KUKA KRL data list: GlobalPosn.dat

&ACCESS RVO1
&REL 1
&PARAM EDITMASK = *
&PARAM TEMPLATE = C:\KRC\Roboter\Template\submit
DEFDAT GlobalPosn PUBLIC
; **************************************
; * Package:     TeslaCore             *
; * Release      V4.0.0                *
; * File:        GlobalPosn.dat        *
; * Date:        07.2016               *
; * GUI Version: > = V8.3              *
; **************************************

;FOLD Control Information
DECL GLOBAL INT nMaxGlobalPosn=10 ; Maximum # of global positions
GLOBAL STRUC PosnCtrl_Typ CHAR Comment[24], BOOL PosnEnabled,AtPosn, INT OutputCtrl, REAL A1_Tol, A2_Tol, A3_Tol, A4_Tol, A5_Tol, A6_Tol, E1_Tol, E2_Tol, E3_Tol, E4_Tol, E5_Tol, E6_Tol
DECL GLOBAL PosnCtrl_Typ xGP_Ctrl[10]
xGP_Ctrl[1]={Comment[]" ", PosnEnabled FALSE, AtPosn FALSE, OutputCtrl 0, A1_Tol 2.0, A2_Tol 2.0, A3_Tol 2.0, A4_Tol 2.0, A5_Tol 2.0, A6_Tol 2.0, E1_Tol 2.0, E2_Tol 2.0, E3_Tol 2.0, E4_Tol 2.0, E5_Tol 2.0, E6_Tol 2.0}
xGP_Ctrl[2]={Comment[]" ", PosnEnabled FALSE, AtPosn FALSE,OutputCtrl 0, A1_Tol 2.0, A2_Tol 2.0, A3_Tol 2.0, A4_Tol 2.0, A5_Tol 2.0, A6_Tol 2.0, E1_Tol 2.0, E2_Tol 2.0, E3_Tol 2.0, E4_Tol 2.0, E5_Tol 2.0, E6_Tol 2.0}
xGP_Ctrl[3]={Comment[]" ", PosnEnabled FALSE, AtPosn FALSE,OutputCtrl 0, A1_Tol 2.0, A2_Tol 2.0, A3_Tol 2.0, A4_Tol 2.0, A5_Tol 2.0, A6_Tol 2.0, E1_Tol 2.0, E2_Tol 2.0, E3_Tol 2.0, E4_Tol 2.0, E5_Tol 2.0, E6_Tol 2.0}
xGP_Ctrl[4]={Comment[]" ", PosnEnabled FALSE, AtPosn FALSE,OutputCtrl 0, A1_Tol 2.0, A2_Tol 2.0, A3_Tol 2.0, A4_Tol 2.0, A5_Tol 2.0, A6_Tol 2.0, E1_Tol 2.0, E2_Tol 2.0, E3_Tol 2.0, E4_Tol 2.0, E5_Tol 2.0, E6_Tol 2.0}
xGP_Ctrl[5]={Comment[]" ", PosnEnabled FALSE, AtPosn FALSE,OutputCtrl 0, A1_Tol 2.0, A2_Tol 2.0, A3_Tol 2.0, A4_Tol 2.0, A5_Tol 2.0, A6_Tol 2.0, E1_Tol 2.0, E2_Tol 2.0, E3_Tol 2.0, E4_Tol 2.0, E5_Tol 2.0, E6_Tol 2.0}
xGP_Ctrl[6]={Comment[]" ", PosnEnabled FALSE, AtPosn FALSE,OutputCtrl 0, A1_Tol 2.0, A2_Tol 2.0, A3_Tol 2.0, A4_Tol 2.0, A5_Tol 2.0, A6_Tol 2.0, E1_Tol 2.0, E2_Tol 2.0, E3_Tol 2.0, E4_Tol 2.0, E5_Tol 2.0, E6_Tol 2.0}
xGP_Ctrl[7]={Comment[]" ", PosnEnabled FALSE, AtPosn FALSE,OutputCtrl 0, A1_Tol 2.0, A2_Tol 2.0, A3_Tol 2.0, A4_Tol 2.0, A5_Tol 2.0, A6_Tol 2.0, E1_Tol 2.0, E2_Tol 2.0, E3_Tol 2.0, E4_Tol 2.0, E5_Tol 2.0, E6_Tol 2.0}
xGP_Ctrl[8]={Comment[]" ", PosnEnabled FALSE, AtPosn FALSE,OutputCtrl 0, A1_Tol 2.0, A2_Tol 2.0, A3_Tol 2.0, A4_Tol 2.0, A5_Tol 2.0, A6_Tol 2.0, E1_Tol 2.0, E2_Tol 2.0, E3_Tol 2.0, E4_Tol 2.0, E5_Tol 2.0, E6_Tol 2.0}
xGP_Ctrl[9]={Comment[]" ", PosnEnabled FALSE, AtPosn FALSE,OutputCtrl 0, A1_Tol 2.0, A2_Tol 2.0, A3_Tol 2.0, A4_Tol 2.0, A5_Tol 2.0, A6_Tol 2.0, E1_Tol 2.0, E2_Tol 2.0, E3_Tol 2.0, E4_Tol 2.0, E5_Tol 2.0, E6_Tol 2.0}
xGP_Ctrl[10]={Comment[]" ", PosnEnabled FALSE, AtPosn FALSE,OutputCtrl 0, A1_Tol 2.0, A2_Tol 2.0, A3_Tol 2.0, A4_Tol 2.0, A5_Tol 2.0, A6_Tol 2.0, E1_Tol 2.0, E2_Tol 2.0, E3_Tol 2.0, E4_Tol 2.0, E5_Tol 2.0, E6_Tol 2.0}
;ENDFOLD (Control Information)
;FOLD Positional Information
DECL GLOBAL E6AXIS XGlobal1={A1 0.0,A2 -90.0,A3 90.0,A4 0.0,A5 0.0,A6 0.0,E1 0.0,E2 0.0,E3 0.0,E4 0.0,E5 0.0,E6 0.0}
DECL GLOBAL FDAT FGlobal1={TOOL_NO 1,BASE_NO 0,IPO_FRAME #BASE,POINT2[] " ",TQ_STATE FALSE}
DECL GLOBAL PDAT PGlobal1={VEL 100.000,ACC 100.000,APO_DIST 100.000,GEAR_JERK 50.0000}
DECL GLOBAL LDAT LCGlobal1={VEL 2.00000,ACC 100.000,APO_DIST 100.000,APO_FAC 50.0000,AXIS_VEL 100.000,AXIS_ACC 100.000,ORI_TYP #VAR,CIRC_TYP #BASE,JERK_FAC 50.0000,GEAR_JERK 50.0000,EXAX_IGN 0}

DECL GLOBAL E6AXIS XGlobal2={A1 0.0,A2 -90.0,A3 90.0,A4 0.0,A5 0.0,A6 0.0,E1 0.0,E2 0.0,E3 0.0,E4 0.0,E5 0.0,E6 0.0}
DECL GLOBAL FDAT FGlobal2={TOOL_NO 1,BASE_NO 0,IPO_FRAME #BASE,POINT2[] " ",TQ_STATE FALSE}
DECL GLOBAL PDAT PGlobal2={VEL 100.000,ACC 100.000,APO_DIST 100.000,GEAR_JERK 50.0000}
DECL GLOBAL LDAT LCGlobal2={VEL 2.00000,ACC 100.000,APO_DIST 100.000,APO_FAC 50.0000,AXIS_VEL 100.000,AXIS_ACC 100.000,ORI_TYP #VAR,CIRC_TYP #BASE,JERK_FAC 50.0000,GEAR_JERK 50.0000,EXAX_IGN 0}

DECL GLOBAL E6AXIS XGlobal3={A1 0.0,A2 -90.0,A3 90.0,A4 0.0,A5 0.0,A6 0.0,E1 0.0,E2 0.0,E3 0.0,E4 0.0,E5 0.0,E6 0.0}
DECL GLOBAL FDAT FGlobal3={TOOL_NO 1,BASE_NO 0,IPO_FRAME #BASE,POINT2[] " ",TQ_STATE FALSE}
DECL GLOBAL PDAT PGlobal3={VEL 100.000,ACC 100.000,APO_DIST 100.000,GEAR_JERK 50.0000}
DECL GLOBAL LDAT LCGlobal3={VEL 2.00000,ACC 100.000,APO_DIST 100.000,APO_FAC 50.0000,AXIS_VEL 100.000,AXIS_ACC 100.000,ORI_TYP #VAR,CIRC_TYP #BASE,JERK_FAC 50.0000,GEAR_JERK 50.0000,EXAX_IGN 0}

DECL GLOBAL E6AXIS XGlobal4={A1 0.0,A2 -90.0,A3 90.0,A4 0.0,A5 0.0,A6 0.0,E1 0.0,E2 0.0,E3 0.0,E4 0.0,E5 0.0,E6 0.0}
DECL GLOBAL FDAT FGlobal4={TOOL_NO 1,BASE_NO 0,IPO_FRAME #BASE,POINT2[] " ",TQ_STATE FALSE}
DECL GLOBAL PDAT PGlobal4={VEL 100.000,ACC 100.000,APO_DIST 100.000,GEAR_JERK 50.0000}
DECL GLOBAL LDAT LCGlobal4={VEL 2.00000,ACC 100.000,APO_DIST 100.000,APO_FAC 50.0000,AXIS_VEL 100.000,AXIS_ACC 100.000,ORI_TYP #VAR,CIRC_TYP #BASE,JERK_FAC 50.0000,GEAR_JERK 50.0000,EXAX_IGN 0}

DECL GLOBAL E6AXIS XGlobal5={A1 0.0,A2 -90.0,A3 90.0,A4 0.0,A5 0.0,A6 0.0,E1 0.0,E2 0.0,E3 0.0,E4 0.0,E5 0.0,E6 0.0}
DECL GLOBAL FDAT FGlobal5={TOOL_NO 1,BASE_NO 0,IPO_FRAME #BASE,POINT2[] " ",TQ_STATE FALSE}
DECL GLOBAL PDAT PGlobal5={VEL 100.000,ACC 100.000,APO_DIST 100.000,GEAR_JERK 50.0000}
DECL GLOBAL LDAT LCGlobal5={VEL 2.00000,ACC 100.000,APO_DIST 100.000,APO_FAC 50.0000,AXIS_VEL 100.000,AXIS_ACC 100.000,ORI_TYP #VAR,CIRC_TYP #BASE,JERK_FAC 50.0000,GEAR_JERK 50.0000,EXAX_IGN 0}

DECL GLOBAL E6AXIS XGlobal6={A1 0.0,A2 -90.0,A3 90.0,A4 0.0,A5 0.0,A6 0.0,E1 0.0,E2 0.0,E3 0.0,E4 0.0,E5 0.0,E6 0.0}
DECL GLOBAL FDAT FGlobal6={TOOL_NO 1,BASE_NO 0,IPO_FRAME #BASE,POINT2[] " ",TQ_STATE FALSE}
DECL GLOBAL PDAT PGlobal6={VEL 100.000,ACC 100.000,APO_DIST 100.000,GEAR_JERK 50.0000}
DECL GLOBAL LDAT LCGlobal6={VEL 2.00000,ACC 100.000,APO_DIST 100.000,APO_FAC 50.0000,AXIS_VEL 100.000,AXIS_ACC 100.000,ORI_TYP #VAR,CIRC_TYP #BASE,JERK_FAC 50.0000,GEAR_JERK 50.0000,EXAX_IGN 0}

DECL GLOBAL E6AXIS XGlobal7={A1 0.0,A2 -90.0,A3 90.0,A4 0.0,A5 0.0,A6 0.0,E1 0.0,E2 0.0,E3 0.0,E4 0.0,E5 0.0,E6 0.0}
DECL GLOBAL FDAT FGlobal7={TOOL_NO 1,BASE_NO 0,IPO_FRAME #BASE,POINT2[] " ",TQ_STATE FALSE}
DECL GLOBAL PDAT PGlobal7={VEL 100.000,ACC 100.000,APO_DIST 100.000,GEAR_JERK 50.0000}
DECL GLOBAL LDAT LCGlobal7={VEL 2.00000,ACC 100.000,APO_DIST 100.000,APO_FAC 50.0000,AXIS_VEL 100.000,AXIS_ACC 100.000,ORI_TYP #VAR,CIRC_TYP #BASE,JERK_FAC 50.0000,GEAR_JERK 50.0000,EXAX_IGN 0}

DECL GLOBAL E6AXIS XGlobal8={A1 0.0,A2 -90.0,A3 90.0,A4 0.0,A5 0.0,A6 0.0,E1 0.0,E2 0.0,E3 0.0,E4 0.0,E5 0.0,E6 0.0}
DECL GLOBAL FDAT FGlobal8={TOOL_NO 1,BASE_NO 0,IPO_FRAME #BASE,POINT2[] " ",TQ_STATE FALSE}
DECL GLOBAL PDAT PGlobal8={VEL 100.000,ACC 100.000,APO_DIST 100.000,GEAR_JERK 50.0000}
DECL GLOBAL LDAT LCGlobal8={VEL 2.00000,ACC 100.000,APO_DIST 100.000,APO_FAC 50.0000,AXIS_VEL 100.000,AXIS_ACC 100.000,ORI_TYP #VAR,CIRC_TYP #BASE,JERK_FAC 50.0000,GEAR_JERK 50.0000,EXAX_IGN 0}

DECL GLOBAL E6AXIS XGlobal9={A1 0.0,A2 -90.0,A3 90.0,A4 0.0,A5 0.0,A6 0.0,E1 0.0,E2 0.0,E3 0.0,E4 0.0,E5 0.0,E6 0.0}
DECL GLOBAL FDAT FGlobal9={TOOL_NO 1,BASE_NO 0,IPO_FRAME #BASE,POINT2[] " ",TQ_STATE FALSE}
DECL GLOBAL PDAT PGlobal9={VEL 100.000,ACC 100.000,APO_DIST 100.000,GEAR_JERK 50.0000}
DECL GLOBAL LDAT LCGlobal9={VEL 2.00000,ACC 100.000,APO_DIST 100.000,APO_FAC 50.0000,AXIS_VEL 100.000,AXIS_ACC 100.000,ORI_TYP #VAR,CIRC_TYP #BASE,JERK_FAC 50.0000,GEAR_JERK 50.0000,EXAX_IGN 0}

DECL GLOBAL E6AXIS XGlobal10={A1 0.0,A2 -90.0,A3 90.0,A4 0.0,A5 0.0,A6 0.0,E1 0.0,E2 0.0,E3 0.0,E4 0.0,E5 0.0,E6 0.0}
DECL GLOBAL FDAT FGlobal10={TOOL_NO 1,BASE_NO 0,IPO_FRAME #BASE,POINT2[] " ",TQ_STATE FALSE}
DECL GLOBAL PDAT PGlobal10={VEL 100.000,ACC 100.000,APO_DIST 100.000,GEAR_JERK 50.0000}
DECL GLOBAL LDAT LCGlobal10={VEL 2.00000,ACC 100.000,APO_DIST 100.000,APO_FAC 50.0000,AXIS_VEL 100.000,AXIS_ACC 100.000,ORI_TYP #VAR,CIRC_TYP #BASE,JERK_FAC 50.0000,GEAR_JERK 50.0000,EXAX_IGN 0}
;ENDFOLD (Positional Information)

ENDDAT
